TYPE ST_Colors :
	STRUCT
		Red	  : BYTE;
		Green : BYTE;
		Blue  : BYTE;
		White : BYTE;
	END_STRUCT
END_TYPE

(* stored: Version 1.1.0.1
   DUT ST_Colors: Id {bb02d163-b628-4acd-b3b4-7e9f50c2410d} *)
